Yaskawa INFORM job: MALBEN1.JBI

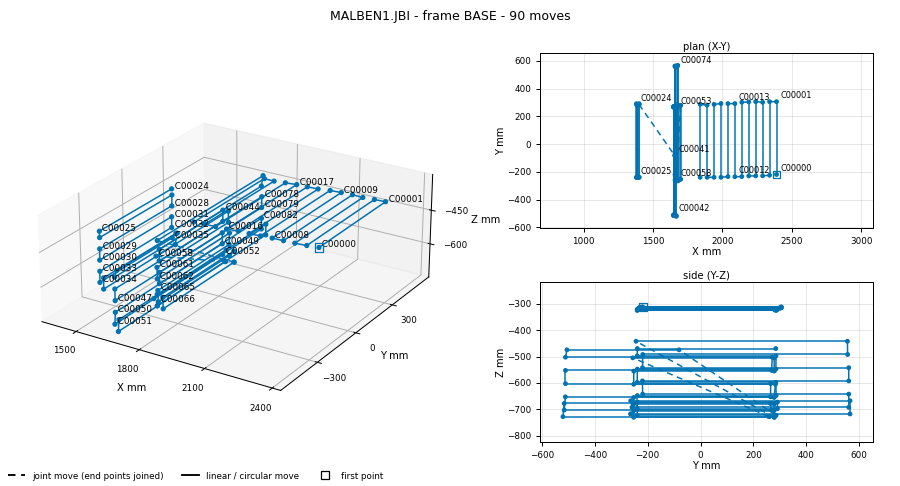
[picture p0: tool path of MALBEN1.JBI in frame BASE, 90 of 96 moves have a stored position in this frame; points joined in program order, loops and branches not executed]
/JOB
//NAME MALBEN1
//POS
///NPOS 90,0,90,0,0,0
///TOOL 0
///POSTYPE BASE
///RECTAN
///RCONF 1,0,0,0,0,0,0,0,0,0,0,0,0,0,0,0,0,0,0,0,0,0,0,0
C00000=2389.234956,-219.082011,-312.004422,175.000000,5.000000,5.000000
C00001=2389.234956,305.508798,-312.004422,175.000000,5.000000,5.000000
C00002=2339.234956,305.593594,-313.482455,175.000000,5.000000,5.000000
C00003=2339.234956,-224.691128,-313.482455,175.000000,5.000000,5.000000
C00004=2289.234956,-228.729284,-314.239196,175.000000,5.000000,5.000000
C00005=2289.234956,300.979638,-314.239196,175.000000,5.000000,5.000000
C00006=2239.234956,305.591915,-315.186482,175.000000,5.000000,5.000000
C00007=2239.234956,-229.178030,-315.186482,175.000000,5.000000,5.000000
C00008=2189.234956,-229.424582,-316.079390,175.000000,5.000000,5.000000
C00009=2189.234956,303.988910,-316.079390,175.000000,5.000000,5.000000
C00010=2139.234956,301.159864,-317.205540,175.000000,5.000000,5.000000
C00011=2139.234956,-233.889375,-317.205540,175.000000,5.000000,5.000000
C00012=2089.234956,-235.160659,-318.373453,175.000000,5.000000,5.000000
C00013=2089.234956,291.489784,-318.373453,175.000000,5.000000,5.000000
C00014=2039.234956,291.425697,-319.682340,175.000000,5.000000,5.000000
C00015=2039.234956,-234.039097,-319.682340,175.000000,5.000000,5.000000
C00016=1989.234956,-239.273769,-321.176978,175.000000,5.000000,5.000000
C00017=1989.234956,291.810217,-321.176978,175.000000,5.000000,5.000000
C00018=1939.234956,285.825535,-322.187816,175.000000,5.000000,5.000000
C00019=1939.234956,-239.273769,-322.187816,175.000000,5.000000,5.000000
C00020=1889.234956,-239.468268,-323.678701,175.000000,5.000000,5.000000
C00021=1889.234956,280.431906,-323.678701,175.000000,5.000000,5.000000
C00022=1839.211746,286.376568,-325.788667,175.000000,5.000000,5.000000
C00023=1839.211746,-239.497932,-325.788667,175.000000,5.000000,5.000000
C00024=1384.941222,284.601818,-469.844109,175.000000,-89.999999,5.000000
C00025=1384.941222,-239.232826,-469.844109,175.000000,-89.999999,5.000000
C00026=1385.410392,-239.430403,-497.715315,175.000000,-89.999999,5.000000
C00027=1385.410392,285.514422,-497.715315,175.000000,-89.999999,5.000000
C00028=1384.099452,285.309289,-547.715315,175.000000,-89.999999,5.000000
C00029=1384.099452,-239.292994,-547.715315,175.000000,-89.999999,5.000000
C00030=1382.905959,-239.589080,-597.715315,175.000000,-89.999999,5.000000
C00031=1382.905959,285.084846,-597.715315,175.000000,-89.999999,5.000000
C00032=1381.752643,285.966387,-647.715315,175.000000,-89.999999,5.000000
C00033=1381.752643,-239.108011,-647.715315,175.000000,-89.999999,5.000000
C00034=1380.544103,-239.108011,-697.715315,175.000000,-89.999999,5.000000
C00035=1380.544103,290.974377,-697.715315,175.000000,-89.999999,5.000000
C00036=1399.775658,290.889301,-672.715315,180.000000,-60.000000,0.000000
C00037=1399.775658,-239.268367,-672.715315,180.000000,-60.000000,0.000000
C00038=1398.985172,-239.728448,-722.715315,180.000000,-60.000000,0.000000
C00039=1398.985172,285.288860,-722.715315,180.000000,-60.000000,0.000000
C00040=1398.985172,285.288860,-722.715315,180.000000,-60.000000,0.000000
C00041=1655.009206,-81.087591,-474.662861,175.000000,-89.999999,5.000000
C00042=1655.009206,-505.623111,-474.662861,175.000000,-89.999999,5.000000
C00043=1648.309269,-511.122524,-502.601943,175.000000,-89.999999,5.000000
C00044=1648.309269,271.097608,-502.601943,175.000000,-89.999999,5.000000
C00045=1648.476917,269.513268,-552.601943,175.000000,-89.999999,5.000000
C00046=1648.476917,-511.123396,-552.601943,175.000000,-89.999999,5.000000
C00047=1648.617373,-511.123396,-602.601943,175.000000,-89.999999,5.000000
C00048=1648.617373,265.347072,-602.601943,175.000000,-89.999999,5.000000
C00049=1648.401920,265.282112,-652.601943,175.000000,-89.999999,5.000000
C00050=1648.401920,-511.551089,-652.601943,175.000000,-89.999999,5.000000
C00051=1648.092484,-515.881648,-702.601943,175.000000,-89.999999,5.000000
C00052=1648.092484,267.925876,-702.601943,175.000000,-89.999999,5.000000
C00053=1667.760043,264.754580,-677.601943,180.000000,-60.000000,0.000000
C00054=1667.760043,-515.882084,-677.601943,180.000000,-60.000000,0.000000
C00055=1667.006814,-520.640335,-727.601943,180.000000,-60.000000,0.000000
C00056=1667.006814,259.465744,-727.601943,180.000000,-60.000000,0.000000
C00057=1667.006814,259.465744,-727.601943,180.000000,-60.000000,0.000000
C00058=1670.020022,-256.322670,-505.109324,175.000000,-89.999999,5.000000
C00059=1670.020022,278.656886,-505.109324,175.000000,-89.999999,5.000000
C00060=1671.157930,278.767988,-555.109324,175.000000,-89.999999,5.000000
C00061=1671.157930,-252.615722,-555.109324,175.000000,-89.999999,5.000000
C00062=1672.503149,-252.957703,-605.109324,175.000000,-89.999999,5.000000
C00063=1672.503149,283.575323,-605.109324,175.000000,-89.999999,5.000000
C00064=1673.920265,278.340371,-655.109324,175.000000,-89.999999,5.000000
C00065=1673.920265,-253.273659,-655.109324,175.000000,-89.999999,5.000000
C00066=1675.302342,-252.957703,-705.109324,175.000000,-89.999999,5.000000
C00067=1675.302342,277.928705,-705.109324,175.000000,-89.999999,5.000000
C00068=1696.826956,278.808007,-680.109324,180.000000,-60.000000,0.000000
C00069=1696.826956,-252.957703,-680.109324,180.000000,-60.000000,0.000000
C00070=1698.068396,-253.117780,-730.109324,180.000000,-60.000000,0.000000
C00071=1698.068396,278.863978,-730.109324,180.000000,-60.000000,0.000000
C00072=1698.068396,278.863978,-730.109324,180.000000,-60.000000,0.000000
C00073=1669.043619,-244.185590,-442.379249,175.000000,-89.999999,5.000000
C00074=1669.043619,555.876896,-442.379249,175.000000,-89.999999,5.000000
C00075=1660.318265,556.650755,-492.379249,175.000000,-89.999999,5.000000
C00076=1660.318265,-218.803450,-492.379249,175.000000,-89.999999,5.000000
C00077=1660.180447,-219.631371,-542.379249,175.000000,-89.999999,5.000000
C00078=1660.180447,560.879731,-542.379249,175.000000,-89.999999,5.000000
C00079=1659.631222,560.881039,-592.379249,175.000000,-89.999999,5.000000
C00080=1659.631222,-219.825816,-592.379249,175.000000,-89.999999,5.000000
C00081=1658.693898,-219.151360,-642.379249,175.000000,-89.999999,5.000000
C00082=1658.693898,560.880603,-642.379249,175.000000,-89.999999,5.000000
C00083=1658.347269,560.937716,-692.379249,175.000000,-89.999999,5.000000
C00084=1658.347269,-259.330556,-692.379249,175.000000,-89.999999,5.000000
C00085=1677.793981,-264.279330,-667.379249,180.000000,-60.000000,0.000000
C00086=1677.793981,565.771392,-667.379249,180.000000,-60.000000,0.000000
C00087=1677.674349,565.782292,-717.379249,180.000000,-60.000000,0.000000
C00088=1677.674349,-264.279330,-717.379249,180.000000,-60.000000,0.000000
C00089=1677.674349,-264.279330,-717.379249,180.000000,-60.000000,0.000000
///POSTYPE PULSE
///PULSE
EC00000=0
EC00001=0
EC00002=0
EC00003=0
EC00004=0
EC00005=0
EC00006=0
EC00007=0
EC00008=0
EC00009=0
EC00010=0
EC00011=0
EC00012=0
EC00013=0
EC00014=0
EC00015=0
EC00016=0
EC00017=0
EC00018=0
EC00019=0
EC00020=0
EC00021=0
EC00022=0
EC00023=0
EC00024=0
EC00025=0
EC00026=0
EC00027=0
EC00028=0
EC00029=0
EC00030=0
EC00031=0
EC00032=0
EC00033=0
EC00034=0
EC00035=0
EC00036=0
EC00037=0
EC00038=0
EC00039=0
EC00040=92160
EC00041=92160
EC00042=92160
EC00043=92160
EC00044=92160
EC00045=92160
EC00046=92160
EC00047=92160
EC00048=92160
EC00049=92160
EC00050=92160
EC00051=92160
EC00052=92160
EC00053=92160
EC00054=92160
EC00055=92160
EC00056=92160
EC00057=184320
EC00058=184320
EC00059=184320
EC00060=184320
EC00061=184320
EC00062=184320
EC00063=184320
EC00064=184320
EC00065=184320
EC00066=184320
EC00067=184320
EC00068=184320
EC00069=184320
EC00070=184320
EC00071=184320
EC00072=276480
EC00073=276480
EC00074=276480
EC00075=276480
EC00076=276480
EC00077=276480
EC00078=276480
EC00079=276480
EC00080=276480
EC00081=276480
EC00082=276480
EC00083=276480
EC00084=276480
EC00085=276480
EC00086=276480
EC00087=276480
EC00088=276480
EC00089=368640
//INST
///DATE 2023/02/06 23:10
///ATTR SC,RW,RJ
////FRAME BASE
///GROUP1 RB1,ST1
NOP
MOVJ P009 EX000 VJ=15.00
MOVJ C00000 EC00000 VJ=15.0
CALL JOB:SPYON
MOVL C00001 EC00001 V=150.0
MOVL C00002 EC00002 V=150.0
MOVL C00003 EC00003 V=150.0
MOVL C00004 EC00004 V=150.0
MOVL C00005 EC00005 V=150.0
MOVL C00006 EC00006 V=150.0
MOVL C00007 EC00007 V=150.0
MOVL C00008 EC00008 V=150.0
MOVL C00009 EC00009 V=150.0
MOVL C00010 EC00010 V=150.0
MOVL C00011 EC00011 V=150.0
MOVL C00012 EC00012 V=150.0
MOVL C00013 EC00013 V=150.0
MOVL C00014 EC00014 V=150.0
MOVL C00015 EC00015 V=150.0
MOVL C00016 EC00016 V=150.0
MOVL C00017 EC00017 V=150.0
MOVL C00018 EC00018 V=150.0
MOVL C00019 EC00019 V=150.0
MOVL C00020 EC00020 V=150.0
MOVL C00021 EC00021 V=150.0
MOVL C00022 EC00022 V=150.0
MOVL C00023 EC00023 V=150.0
CALL JOB:SPYOF
MOVJ P009 VJ=15.00
MOVJ C00024 EC00024 VJ=15.0
CALL JOB:SPYON
MOVL C00025 EC00025 V=150.0
MOVL C00026 EC00026 V=150.0
MOVL C00027 EC00027 V=150.0
MOVL C00028 EC00028 V=150.0
MOVL C00029 EC00029 V=150.0
MOVL C00030 EC00030 V=150.0
MOVL C00031 EC00031 V=150.0
MOVL C00032 EC00032 V=150.0
MOVL C00033 EC00033 V=150.0
MOVL C00034 EC00034 V=150.0
MOVL C00035 EC00035 V=150.0
MOVL C00036 EC00036 V=150.0
MOVL C00037 EC00037 V=150.0
MOVL C00038 EC00038 V=150.0
MOVL C00039 EC00039 V=150.0
CALL JOB:SPYOF
MOVJ P009 VJ=15.00
MOVL C00040 EC00040 V=150.0
MOVJ C00041 EC00041 VJ=15.0
CALL JOB:SPYON
MOVL C00042 EC00042 V=150.0
MOVL C00043 EC00043 V=150.0
MOVL C00044 EC00044 V=150.0
MOVL C00045 EC00045 V=150.0
MOVL C00046 EC00046 V=150.0
MOVL C00047 EC00047 V=150.0
MOVL C00048 EC00048 V=150.0
MOVL C00049 EC00049 V=150.0
MOVL C00050 EC00050 V=150.0
MOVL C00051 EC00051 V=150.0
MOVL C00052 EC00052 V=150.0
MOVL C00053 EC00053 V=150.0
MOVL C00054 EC00054 V=150.0
MOVL C00055 EC00055 V=150.0
MOVL C00056 EC00056 V=150.0
CALL JOB:SPYOF
MOVJ P009 VJ=15.00
MOVL C00057 EC00057 V=150.0
MOVJ C00058 EC00058 VJ=15.0
CALL JOB:SPYON
MOVL C00059 EC00059 V=150.0
MOVL C00060 EC00060 V=150.0
MOVL C00061 EC00061 V=150.0
MOVL C00062 EC00062 V=150.0
MOVL C00063 EC00063 V=150.0
MOVL C00064 EC00064 V=150.0
MOVL C00065 EC00065 V=150.0
MOVL C00066 EC00066 V=150.0
MOVL C00067 EC00067 V=150.0
MOVL C00068 EC00068 V=150.0
MOVL C00069 EC00069 V=150.0
MOVL C00070 EC00070 V=150.0
MOVL C00071 EC00071 V=150.0
CALL JOB:SPYOF
MOVJ P009 VJ=15.00
MOVL C00072 EC00072 V=150.0
MOVJ C00073 EC00073 VJ=15.0
CALL JOB:SPYON
MOVL C00074 EC00074 V=150.0
MOVL C00075 EC00075 V=150.0
MOVL C00076 EC00076 V=150.0
MOVL C00077 EC00077 V=150.0
MOVL C00078 EC00078 V=150.0
MOVL C00079 EC00079 V=150.0
MOVL C00080 EC00080 V=150.0
MOVL C00081 EC00081 V=150.0
MOVL C00082 EC00082 V=150.0
MOVL C00083 EC00083 V=150.0
MOVL C00084 EC00084 V=150.0
MOVL C00085 EC00085 V=150.0
MOVL C00086 EC00086 V=150.0
MOVL C00087 EC00087 V=150.0
MOVL C00088 EC00088 V=150.0
CALL JOB:SPYOF
MOVJ P009 VJ=15.00
MOVL C00089 EC00089 V=150.0
END
